PROGRAM MAIN
VAR
	fbKVM: FB_KVM;
	fbCartesian: Cartesian;
END_VAR

fbKVM(wAID:=1 );

fbCartesian(
	boEnable:=INPUT.iboEmergencyStopBut , 
	boStartAck=> , 	
	boEnabAck=> );

END_PROGRAM

(* stored: Version 1.1.0.1, ProductVersion 3.1.4024.12
   POU MAIN: Id {17fb778a-02bd-4788-a0ad-2e1686ce558b}, SpecialFunc None *)
